FUNCTION_BLOCK FB_Z_Axis_TargetPositionConvert
VAR_INPUT
	lrX_AxisTP		:LREAL;	(*X軸のターゲットポジション*)
	lrY_AxisTP		:LREAL;	(*Y軸のターゲットポジション*)
	lrZ_AxisTP		:LREAL;	(*Z軸のターゲットポジション*)
END_VAR
VAR_OUTPUT
	lrZ_AxisConTP	:LREAL;	(*調整後のZ軸のターゲットポジション*)
END_VAR
VAR
	lrXbuf			:LREAL;
	lrYbuf			:LREAL;
END_VAR

	lrXbuf:=GVL.lrXZ_Slope*lrX_AxisTP;
	lrYbuf:=GVL.lrYZ_Slope*lrY_AxisTP;
	
	lrZ_AxisConTP:=lrZ_AxisTP+lrXbuf+lrYbuf;

END_FUNCTION_BLOCK

(* stored: Version 1.1.0.1, ProductVersion 3.1.4026.11
   POU FB_Z_Axis_TargetPositionConvert: Id {a4b216e6-5f91-43c0-9777-25764d252227}, SpecialFunc None *)
